# EPICS autosave request: iocBoot/iocUSBCTR/auto_settings.req
file "USBCTR_settings.req", P=$(P), MP=$(MP)
